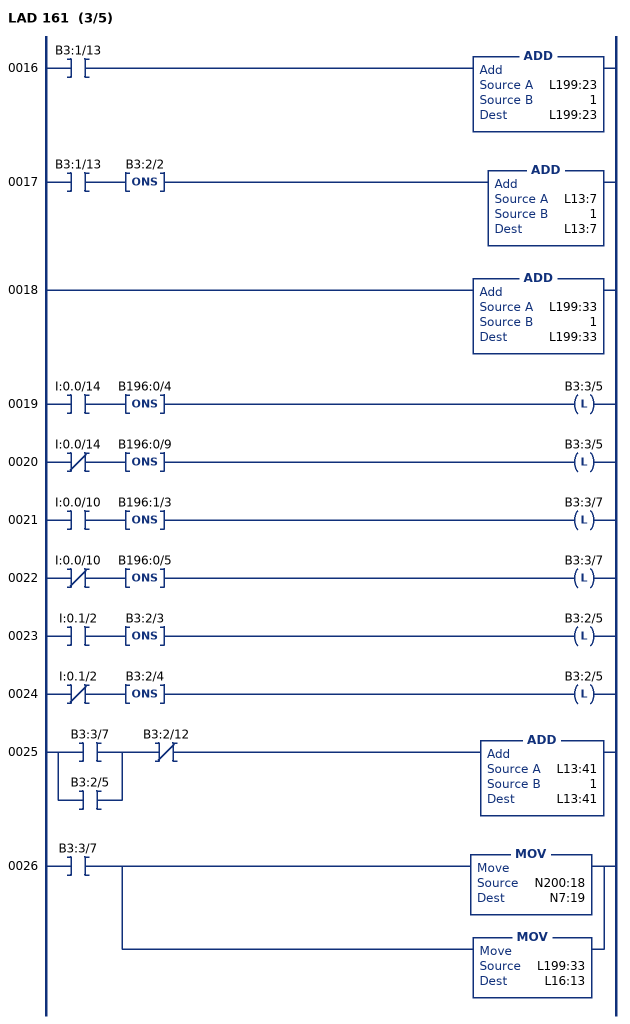
% Rung: 16 %
SOR XIC B3:1/13 ADD L199:23 1 L199:23 EOR
% Rung: 17 %
SOR XIC B3:1/13 ONS B3:2/2 ADD L13:7 1 L13:7 EOR
% Rung: 18 %
SOR ADD L199:33 1 L199:33 EOR
% Rung: 19 %
SOR XIC I:0.0/14 ONS B196:0/4 OTL B3:3/5 EOR
% Rung: 20 %
SOR XIO I:0.0/14 ONS B196:0/9 OTL B3:3/5 EOR
% Rung: 21 %
SOR XIC I:0.0/10 ONS B196:1/3 OTL B3:3/7 EOR
% Rung: 22 %
SOR XIO I:0.0/10 ONS B196:0/5 OTL B3:3/7 EOR
% Rung: 23 %
SOR XIC I:0.1/2 ONS B3:2/3 OTL B3:2/5 EOR
% Rung: 24 %
SOR XIO I:0.1/2 ONS B3:2/4 OTL B3:2/5 EOR
% Rung: 25 %
SOR BST XIC B3:3/7 NXB XIC B3:2/5 BND XIO B3:2/12 ADD L13:41 1 L13:41 EOR
% Rung: 26 %
SOR XIC B3:3/7 BST MOV N200:18 N7:19 NXB MOV L199:33 L16:13 BND EOR

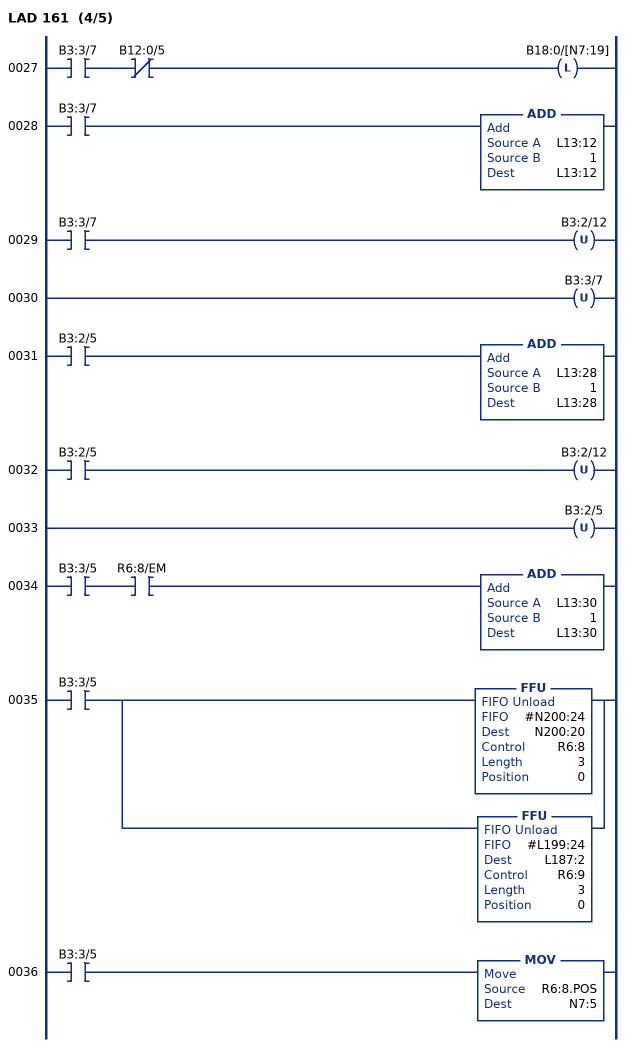
% Rung: 27 %
SOR XIC B3:3/7 XIO B12:0/5 OTL B18:0/[N7:19] EOR
% Rung: 28 %
SOR XIC B3:3/7 ADD L13:12 1 L13:12 EOR
% Rung: 29 %
SOR XIC B3:3/7 OTU B3:2/12 EOR
% Rung: 30 %
SOR OTU B3:3/7 EOR
% Rung: 31 %
SOR XIC B3:2/5 ADD L13:28 1 L13:28 EOR
% Rung: 32 %
SOR XIC B3:2/5 OTU B3:2/12 EOR
% Rung: 33 %
SOR OTU B3:2/5 EOR
% Rung: 34 %
SOR XIC B3:3/5 XIC R6:8/EM ADD L13:30 1 L13:30 EOR
% Rung: 35 %
SOR XIC B3:3/5 BST FFU #N200:24 N200:20 R6:8 3 0 NXB FFU #L199:24 L187:2 R6:9 3 0 BND EOR
% Rung: 36 %
SOR XIC B3:3/5 MOV R6:8.POS N7:5 EOR

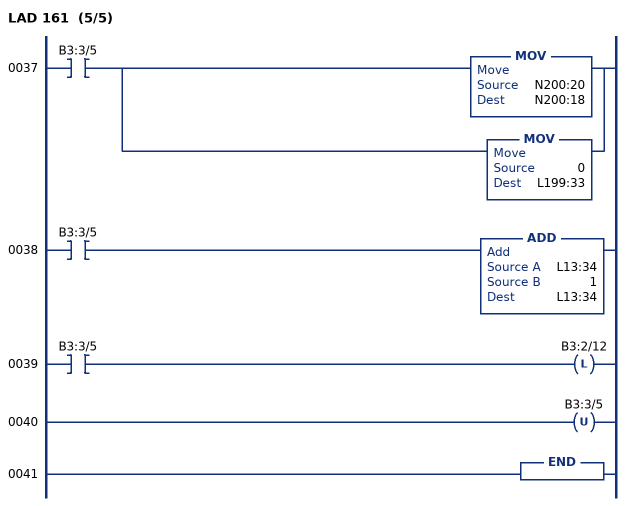
% Rung: 37 %
SOR XIC B3:3/5 BST MOV N200:20 N200:18 NXB MOV 0 L199:33 BND EOR
% Rung: 38 %
SOR XIC B3:3/5 ADD L13:34 1 L13:34 EOR
% Rung: 39 %
SOR XIC B3:3/5 OTL B3:2/12 EOR
% Rung: 40 %
SOR OTU B3:3/5 EOR
% Rung: 41 %
SOR END EOR

LADDER 170
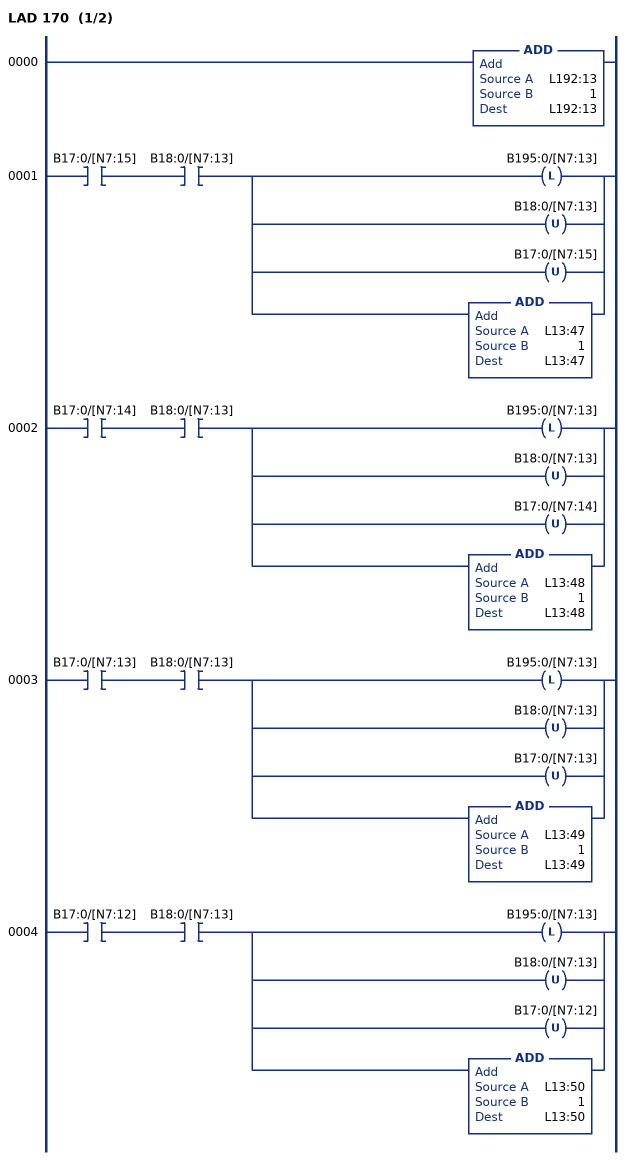
% Rung: 0 %
SOR ADD L192:13 1 L192:13 EOR
% Rung: 1 %
SOR XIC B17:0/[N7:15] XIC B18:0/[N7:13] BST OTL B195:0/[N7:13] NXB OTU B18:0/[N7:13] NXB OTU B17:0/[N7:15] NXB ADD L13:47 1 L13:47 BND EOR
% Rung: 2 %
SOR XIC B17:0/[N7:14] XIC B18:0/[N7:13] BST OTL B195:0/[N7:13] NXB OTU B18:0/[N7:13] NXB OTU B17:0/[N7:14] NXB ADD L13:48 1 L13:48 BND EOR
% Rung: 3 %
SOR XIC B17:0/[N7:13] XIC B18:0/[N7:13] BST OTL B195:0/[N7:13] NXB OTU B18:0/[N7:13] NXB OTU B17:0/[N7:13] NXB ADD L13:49 1 L13:49 BND EOR
% Rung: 4 %
SOR XIC B17:0/[N7:12] XIC B18:0/[N7:13] BST OTL B195:0/[N7:13] NXB OTU B18:0/[N7:13] NXB OTU B17:0/[N7:12] NXB ADD L13:50 1 L13:50 BND EOR

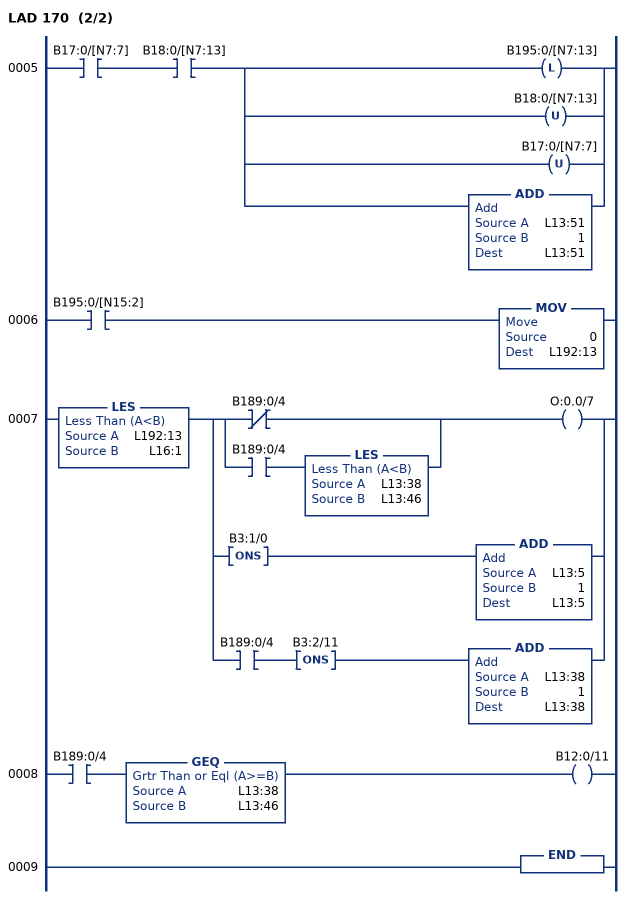
% Rung: 5 %
SOR XIC B17:0/[N7:7] XIC B18:0/[N7:13] BST OTL B195:0/[N7:13] NXB OTU B18:0/[N7:13] NXB OTU B17:0/[N7:7] NXB ADD L13:51 1 L13:51 BND EOR
% Rung: 6 %
SOR XIC B195:0/[N15:2] MOV 0 L192:13 EOR
% Rung: 7 %
SOR LES L192:13 L16:1 BST BST XIO B189:0/4 NXB XIC B189:0/4 LES L13:38 L13:46 BND OTE O:0.0/7 NXB ONS B3:1/0 ADD L13:5 1 L13:5 NXB XIC B189:0/4 ONS B3:2/11 ADD L13:38 1 L13:38 BND EOR
% Rung: 8 %
SOR XIC B189:0/4 GEQ L13:38 L13:46 OTE B12:0/11 EOR
% Rung: 9 %
SOR END EOR

LADDER 180
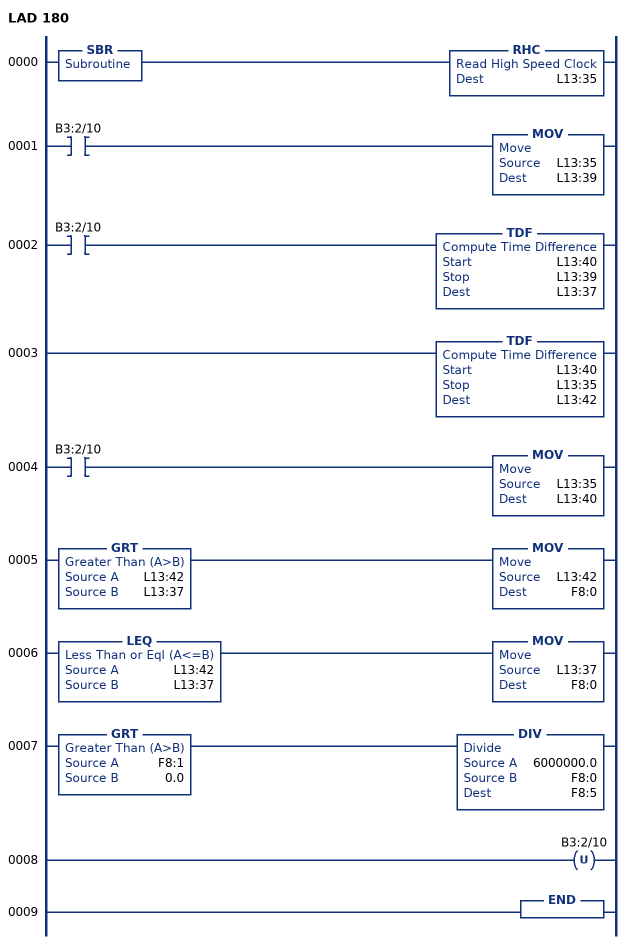
% Rung: 0 %
SOR SBR RHC L13:35 EOR
% Rung: 1 %
SOR XIC B3:2/10 MOV L13:35 L13:39 EOR
% Rung: 2 %
SOR XIC B3:2/10 TDF L13:40 L13:39 L13:37 EOR
% Rung: 3 %
SOR TDF L13:40 L13:35 L13:42 EOR
% Rung: 4 %
SOR XIC B3:2/10 MOV L13:35 L13:40 EOR
% Rung: 5 %
SOR GRT L13:42 L13:37 MOV L13:42 F8:0 EOR
% Rung: 6 %
SOR LEQ L13:42 L13:37 MOV L13:37 F8:0 EOR
% Rung: 7 %
SOR GRT F8:1 0.0 DIV 6000000.0 F8:0 F8:5 EOR
% Rung: 8 %
SOR OTU B3:2/10 EOR
% Rung: 9 %
SOR END EOR

DATA TABLE (non-zero values as saved)
DATA B3
% B3:0 % 0X8021 0X0050 0X8090 0XA200 0X0306 0X2000 0X02C1 0X0020 0X4007 0X0000
% B3:10 % 0X2041 0X0846 0X2000 0X0000
DATA T4
% .PRE .ACC %
% T4:0 % 300 0
% T4:1 % 150 152
% T4:2 % 32765 0
% T4:3 % 32765 0
% T4:4 % 32765 0
% T4:5 % 150 150
% T4:6 % 5555 0
% T4:7 % 10 0
% T4:8 % 300 0
% T4:9 % 30 0
% T4:10 % 35 0
% T4:12 % 50 0
% T4:13 % 222 0
% T4:14 % 222 0
% T4:15 % 180 0
% T4:16 % 222 0
% T4:17 % 300 0
% T4:18 % 8 0
% T4:19 % 6 0
% T4:20 % 10 0
% T4:21 % 100 0
% T4:22 % 20 0
% T4:23 % 900 0
% T4:24 % 1000 0
% T4:25 % 250 250
% T4:26 % 666 666
% T4:27 % 400 0
% T4:28 % 400 0
% T4:29 % 10 0
% T4:30 % 50 50
% T4:31 % 20 0
% T4:32 % 69 0
DATA R6
% .LEN .POS %
% R6:0 % 3 0
% R6:1 % 3 0
% R6:2 % 3 0
% R6:3 % 3 0
% R6:4 % 2048 0
% R6:5 % 2048 0
% R6:6 % 912 0
% R6:7 % 435 0
% R6:8 % 3 0
% R6:9 % 3 0
% R6:10 % 659 0
% R6:11 % 659 0
% R6:12 % 2048 0
DATA N7
% N7:0 % 6 1224 0 996 0 0 1 1611 92 75
% N7:10 % 1216 61 1610 1609 1608 1607 3 3 1219 1235
% N7:20 % 0 0 0 0 0 0 -403 0 0 0
% N7:50 % 1236 0 175 16 0 0 0 1464 12 0
% N7:60 % 1 32767 4012 20 31 0 0 15 30 20
% N7:70 % 0 21 23 27738 32767 0 122 0 16 0
% N7:80 % 0 6 95 0 0 0 5 500 0 0
% N7:90 % 2011 4 4 12 1 0 0 0 0 1600
% N7:100 % 123 124 1227 1228 1237 1238 0 0 0 0
% N7:110 % 0 0 0 0 0 0 0 0 400 0
% N7:120 % 25007 61 0 0 0 0 0 0 0 0
DATA F8
% F8:0 % 4.805587e+08 206.64 0.20664 5.736945e-05 17430.88
% F8:5 % 0.01248547 0 0 0 198
% F8:10 % 0.0888 0.08897486 2235 101 63.26563
% F8:15 % 37.73437 4040 198 0 0
% F8:20 % 0 0.02 0 1 0
% F8:25 % 0 932781 0.222 279.6551 848597
% F8:30 % 0 170 0.03 38 852060
% F8:35 % 0 0 0 0 77
% F8:40 % 101 37.73437 0 100 1
% F8:45 % 1 2 0.21455 0 0
% F8:50 % 0 0 1 0 1
% F8:55 % 2000000 -221 0 0 0
% F8:95 % 0 0 0 492 4.92
DATA B9
% B9:130 % 0X0000 0X0000 0X0000 0X0000 0X2000 0X0000 0X0000 0X0000 0X0000 0X8000
% B9:140 % 0X2480 0X0000 0X0000 0X0000 0X0000 0X0000 0X0000 0X0000 0X0000 0X0000
% B9:160 % 0X0000 0X0000 0X0000 0X0000 0X0000 0X0000 0X2000 0X0002 0X0000 0X0000
% B9:170 % 0X0000 0X0000 0X0000 0X2000 0X0000 0X0000 0X0000 0X0000 0X0000 0X0000
% B9:180 % 0X0000 0X0000 0X0000 0X0000 0X0000 0X0002 0X0000 0X0000 0X0000 0X0000
% B9:190 % 0X0010 0X0000 0X0000 0X0000 0X0000 0X0000 0X0000 0X0000 0X0000 0X0000
% B9:200 % 0X2B64 0X2B64 0X0000 0X0010 0X0000 0X2000 0X0000 0X0000 0X0000 0X0000
% B9:220 % 0X0000 0X0000 0X0000 0X0200 0X0000 0X0000 0X0000 0X0000 0X0000 0X0020
% B9:230 % 0X0040 0X0000 0X0000 0X0000 0X0000 0X0000 0X0000 0X0000 0X0000 0X0000
DATA B11
% B11:180 % 0X0000 0X8000 0X0000 0X0000 0X0000 0X0000 0X0000 0X0000 0X0000 0X0000
% B11:240 % 0X0000 0X0000 0X0000 0X4000 0X0000 0X0000 0X0000 0X0000 0X0000 0X0000
DATA B12
% B12:0 % 0X01D5 0X0000 0X0000 0X0000 0X0000 0X0000 0X0000 0X0000 0X0000 0X0000
DATA L13
% L13:0 % 308402300 308407124 4824 0 1000
% L13:5 % 296119 12 7 1162124017 1162124017
% L13:10 % 492 308458 310348 323451 323257
% L13:15 % 0 0 0 2147483647 82058
% L13:25 % 0 0 0 13093 14784
% L13:30 % 126 129 323242 99 323441
% L13:35 % 159884200 454 1821512 0 -320753228
% L13:40 % -320753228 434 480641256 802676 29196
% L13:45 % 740408 100 9 5 4716071
% L13:50 % 6 5 2147483647 0 0
DATA F14
% F14:0 % 270.6707 269.8895 27 27 1408.938
% F14:5 % 9502.14 13106.4 982.98 0 0
DATA N15
% N15:0 % 6 908 1612 1224 1212 170 101 1204 1004 5555
% N15:10 % 62 620 0 0 0 0 1204 0 0 0
DATA L16
% L16:0 % 8 9 5 5 5
% L16:5 % 250 5000 5000 192 20
% L16:10 % 1256 1 2045 1 98
% L16:15 % 99 0 0 0 0
DATA B17
% B17:100 % 0X0000 0X0000 0X0000 0X0000 0X0000 0X0000 0X0800 0X0000 0X1000 0X0000
% B17:110 % 0X4000 0X0000 0X0000 0X0000 0X0000 0X0000 0X0000 0X0000 0X0000 0X0000
% B17:120 % 0X0000 0X0000 0X0000 0X0000 0X0000 0X0000 0X0000 0X2000
DATA B18
% B18:100 % 0X0000 0X0000 0X0000 0X0000 0X0000 0X0001 0X0000 0X0080 0X0000 0X8240
% B18:110 % 0X0000 0X0400 0X0000 0X0000 0X0000 0X0000 0X0040 0X0000 0X0000 0X0010
% B18:120 % 0X0000 0X0000 0X0000 0X0000 0X0000 0X0000 0X0000 0X2000
DATA L23
% L23:0 % 65535 -65536 -65536 -65536 -65536
% L23:5 % -65536 -65536 198 65535 -65536
% L23:10 % -65536 0 17 10 17
% L23:15 % 0 0 0 0 8
% L23:20 % 0 -65536 -65536 -65536 -65536
% L23:25 % -65536 20 19 20 0
% L23:30 % 0 0 -65536 -65536 -65536
% L23:35 % -65536 -65536 -65536 -65536 -65536
% L23:40 % 16270 18414 0 63266 -65536
% L23:45 % 5062 0 0 0 0
% L23:50 % 0 -65536 -65536 17 -65536
% L23:55 % 33 5079 -65536 0 0
% L23:60 % 0 -65536 -65536 -65536 0
DATA L24
% L24:0 % -65536 122 -65536 222 -65536
% L24:5 % 65535 -65536 -65536 -65536 -65536
% L24:10 % 50 27 0 1 23
% L24:15 % 1198 1030 95 18 30
% L24:20 % 30 -65536 1226 -65536 -65536
% L24:25 % 222 1236 -65536 -65536 222
% L24:30 % 1466 27 10000 -65536 55
% L24:35 % 180 -65536 180 65535 101
% L24:40 % 101 1000 -65536 -65536 10
% L24:45 % 222 192 -65536 0 -65536
% L24:50 % -999 30 10000 65535 900
DATA L42
% L42:0 % -65536 0 0 0 0
% L42:5 % 45 45 45 0 0
% L42:20 % 0 0 32766 32766 0
% L42:50 % 0 30
DATA L183
% L183:0 % 999 216325420 12 1000000000 0
% L183:5 % 37 48 55 0 0
DATA B185
% B185:0 % 0X0200 0X0001 0X0000 0X0000 0X0000 0X0000 0X0000 0X0000 0X0000 0X0000
DATA N186
% N186:0 % 100 0 0 0 0 0 0 0 0 0
DATA L187
% L187:0 % 65 23 37 0 0
% L187:5 % 1063 0 0 0 0
DATA F188
% F188:0 % 6 66 11 44 29
DATA B189
% B189:0 % 0X00E0 0X0000 0X0000 0X0000 0X0000 0X0000 0X0000 0X0000 0X0000 0X0000
DATA L190
% L190:0 % 1 5 0 0 0
% L190:30 % 0 2 0 0 0
DATA B191
% B191:0 % 0X0000 0X0001 0X0000 0X0000 0X0000 0X0000 0X0000 0X0000 0X0000 0X0000
DATA L192
% L192:0 % 160119659 160119659 369 118 43694
% L192:5 % 100000 13600000 999 999 8
% L192:10 % 0 0 0 1297767 17
% L192:15 % 160119564 160119564 372 117 43326
% L192:20 % 180 13700000 0 0 0
DATA F193
% F193:0 % 1.002432 0.315 0.022 6 270
% F193:5 % -0.2756042 0.15 -0.04134064 270.6568 8868.34
% F193:10 % 0.011 0.195 0.165 0.337 270
% F193:15 % 0.008728027 0.15 0.001309204 346.8937 11366.32
DATA B195
% B195:60 % 0X0000 0X0000 0X0000 0X0000 0X0000 0X0000 0X0000 0X0000 0X4000 0X19C0
% B195:70 % 0X8000 0X84B0 0X0210 0X0000 0X0000 0X0000 0X0000 0X0000 0X0000 0X0000
DATA B196
% B196:0 % 0X0A27 0X9FF2 0X0005 0X0000 0X0000 0X0000 0X0000 0X0000 0X0000 0X0000
% B196:30 % 0XE800 0X9BFF 0XEBFF 0XFFDF 0XFFFF 0X0000 0X0000 0X0000 0X0000 0X0000
DATA N197
% N197:0 % 1560 150 1111 2500 2500 14417 5555 300 150 0
% N197:10 % 4000 969 4 0 0 0 0 0 0 0
% N197:30 % 15 48 0 0 0 0 0 0 0 0
DATA B198
% B198:0 % 0X0009 0X0000 0X0000 0X0000 0X0000 0X0000 0X0000 0X0000 0X0000 0X0000
DATA L199
% L199:0 % 1 5571998 134 11 3579521
% L199:5 % 0 0 0 5 174974
% L199:10 % 0 224 10256 112 0
% L199:15 % 0 0 0 278717848 518
% L199:20 % 4767338 16430853 5001 5001 0
% L199:25 % 0 0 3890781 999 4770366
% L199:30 % 4770321 251 4553523 4553523 111
% L199:35 % 555 555 0 0 0
DATA N200
% N200:0 % 2046 2047 2046 2047 2045 200 1006 2045 2045 2045
% N200:10 % 0 0 0 1277 187 2046 1000 2045 2045 1218
% N200:20 % 1234 0 0 0 0 0 0 0 0 0
% N200:30 % 0 0 32767 0 0 0 0 0 0 0
DATA L201
% L201:0 % 20 40 40 -3011735 44
% L201:5 % 96629277 0 0 -3010662 0
% L201:10 % 0 0 0 327 43
% L201:15 % 0 43 0 43 36830
DATA B202
% B202:0 % 0X2241 0X0000 0X0001 0X0000 0X0000 0X0000 0X0000 0X0000 0X0000 0X0000
DATA N203
% N203:0 % 115 115 116 333 334 333 444 0 445 444
% N203:10 % 555 556 555 0 0 0 0 0 0 0
DATA L204
% L204:0 % 111 101 111 18068 89006
% L204:5 % 0 0 18069 222 0
% L204:10 % 0 0 0 1327077052 1327077052
% L204:15 % 1327077052 1327077052 1 0 0
% L204:20 % 0 0 33 0 0
% L204:30 % 33 0 0 0 0
DATA F205
% F205:0 % 655.32 655.32 655.32 655.32 0
